(* IEC 61131-3 sources: AXOpen/src/io/ctrl/src, 12 files *)

(* ---- ComponentAvailability.st ---- *)
NAMESPACE AXOpen.Io
    TYPE ComponentAvailability : UINT (
        Available	            :=  UINT#0,	// Hardware component is available.
        ApplicationReadyPending	:=  UINT#1,	// Application Ready Pending; no I/O access.
        LockedBySuperordinated	:=  UINT#2,	// Locked by Superordinated; no access to hardware component.
        LockedByIOController	:=  UINT#3,	// Locked by IO controller; no access to hardware component.
        LockedByIOSupervisor	:=  UINT#4	// Locked by IO supervisor; no access to hardware component.
    );
    END_TYPE
END_NAMESPACE

(* ---- ComponentState.st ---- *)
NAMESPACE AXOpen.Io
    TYPE ComponentState  : UINT (
        Good                    :=	UINT#0, //	No problems detected.
        Disabled                :=	UINT#1, //	The hardware component is disabled.
        MaintenanceRequired     :=	UINT#2, //	Maintenance required.
        MaintenanceDemanded     :=	UINT#3, //	Maintenance demanded.
        Error                   :=	UINT#4, //	Error.
        NotAccessible           :=	UINT#5, //	Status unknown or error in higher-level hardware component.
        Unknown                 :=	UINT#6, //	Default value for components that do not return diagnostic events.
        IONotAvailable          :=	UINT#7  //	Inputs/outputs are not available.
                    );
    END_TYPE
END_NAMESPACE

(* ---- GetDiagnosticsReturnCode.st ---- *)
NAMESPACE AXOpen.Io
    TYPE GetDiagnosticsReturnCode : INT (
        Unknown             :=	INT#-1,     //
        NoError             :=	INT#0,      //	No error.
        HardwareIDInvalid   :=	INT#-32642, //	The address is unknown.
        HardwareIDisInvalid   :=	INT#-32624, //	The address is unknown.
        OutOfResources      :=	INT#-32575  //	All diagnostic resources are currently in use
        ) := Unknown;
    END_TYPE
END_NAMESPACE

(* ---- OperatingState .st ---- *)
NAMESPACE AXOpen.Io
    TYPE OperatingState   : UINT (
        NotSupported                :=	UINT#0,     //	Not Supported; for I/O modules OperatingState always has this value.
        StopFirmwareUpdate          :=	UINT#1,     //	STOP; firmware update.
        StopMemoryReset             :=	UINT#2,     //	STOP; memory reset.
        StopSelfStart               :=	UINT#3,     //	STOP; self start.
        Stop                        :=	UINT#4,     //	STOP.
        MemoryReset                 :=	UINT#5,     //	Memory reset.
        Startup                     :=	UINT#6,     //	STARTUP.
        Run                         :=	UINT#8,     //	RUN.
        RunRedundant                :=	UINT#9,     //	RUN-REDUNDANT.
        Hold                        :=	UINT#10,    //	HOLD.
        Defect                      :=	UINT#13,    //	DEFECT (can only be seen in diagnostic buffer entries).
        DeEnergized                 :=	UINT#15,    //	De-energized (can only be seen in diagnostic buffer entries).
        ConfigurationInRun          :=	UINT#16,    //	Configuration in Run (CiR).
        StopWithoutOutputDisable    :=	UINT#17,    //	STOP without output disable.
        RunWithOutputDisable        :=	UINT#18,    //	RUN with output disable.
        PgmTest                     :=	UINT#19,    //	PgmTest.
        PrimaryRunBackupTest        :=	UINT#20,    //	RunPgmTest (state of primary PLC when the backup PLC is in test mode).
        PrimarySyncup               :=	UINT#21,    //	RUN-SYNCUP (only primary PLC in SYNCUP system state).
        BackupSyncup                :=	UINT#22,    //	SYNCUP (only backup PLC in SYNCUP system state)
        PartnerPlcStateUnknown      :=	UINT#31,    //	State of partner PLC unknown (for example when the partner PLC is not available).
        StopSystemState             :=	UINT#33,    //	STOP system state
        StartupSystemState          :=	UINT#35,    //	STARTUP system state
        RunSoloSystemState          :=	UINT#37,    //	RUN-SOLO system state
        SyncupSystemState           :=	UINT#38,    //	SYNCUP system state
        RunRedundantSystemState     :=	UINT#40    //	RUN-REDUNDANT system state
                    );
    END_TYPE
END_NAMESPACE

(* ---- ReplacementState .st ---- *)
NAMESPACE AXOpen.Io
    TYPE ReplacementState  : UINT (
        Unknown         :=	UINT#255,
        OK              :=	UINT#0, //	The correct element exists.
        Substitute      :=	UINT#1, //	The element was replaced by a compatible element.
        Incompatible    :=	UINT#2, //	The element was replaced by an incompatible element (is reachable, but not ready for operation).
        Missing         :=	UINT#3 //	The element does not exist.
            ) := Unknown;
    END_TYPE
END_NAMESPACE

(* ---- AxoHardwareDiagnostics.st ---- *)
USING AXOpen.Core;
USING AXOpen.Core;
USING AXOpen.Messaging;
USING AXOpen.Messaging.Static;
USING Siemens.Simatic.Diagnostics.Hardware;

NAMESPACE AXOpen.Io
    {S7.extern=ReadWrite}
    CLASS AxoHardwareDiagnostics EXTENDS AXOpen.Core.AxoTask
        VAR PUBLIC
            {#ix-attr:[Container(Layout.Stack)]}
            {#ix-set:AttributeName = "<#Hardware ID#>"}
            {#ix-attr:[ReadOnly()]}
            hardwareID	                :   UINT;	                //  Input	Hardware identifier of the component.
            {#ix-set:AttributeName = "<#Diagnostics return code#>"}
            {#ix-attr:[ReadOnly()]}
            GetDiagnosticsReturnCode    :   GetDiagnosticsReturnCode;
            {#ix-attr:[Container(Layout.Wrap)]}
            {#ix-set:AttributeName = "<#Diagnostics details#>"}
            {#ix-attr:[ReadOnly()]}
            diagnosticDetails	        :   DiagnosticDetails;	    //  Diagnostic information of the addressed hardware component.
        END_VAR

        ///<summary>
        /// Runs tasks and logic of this component.
        /// >[!IMPORTANT] This method must or one of its overloads be called cyclically.
        ///</summary>
        METHOD PUBLIC Run
            VAR_INPUT
                inParent    :   IAxoObject;
                hwID        :   UINT;
            END_VAR
            VAR
                diagInfo : Siemens.Simatic.Diagnostics.Hardware.DiagnosticDetails;
            END_VAR

            IF SUPER.Execute(inParent) THEN
                GetDiagnosticsReturnCode := GetDiagnostics(hwID, diagInfo);

                IF GetDiagnosticsReturnCode=GetDiagnosticsReturnCode#NoError THEN
                    diagnosticDetails.ComponentStateDetail.HardwareComponentState.NoAdditionalInformation   :=  diagInfo.ComponentStateDetail.HardwareComponentState.NoAdditionalInformation;
                    diagnosticDetails.ComponentStateDetail.HardwareComponentState.TransferNotPermitted      :=  diagInfo.ComponentStateDetail.HardwareComponentState.TransferNotPermitted;
                    diagnosticDetails.ComponentStateDetail.HardwareComponentState.DiagnosticsAvailable      :=  diagInfo.ComponentStateDetail.HardwareComponentState.DiagnosticsAvailable;
                    diagnosticDetails.ComponentStateDetail.HardwareComponentState.MaintenanceRequired       :=  diagInfo.ComponentStateDetail.HardwareComponentState.MaintenanceRequired;
                    diagnosticDetails.ComponentStateDetail.HardwareComponentState.MaintenanceDemanded       :=  diagInfo.ComponentStateDetail.HardwareComponentState.MaintenanceDemanded;
                    diagnosticDetails.ComponentStateDetail.HardwareComponentState.Error                     :=  diagInfo.ComponentStateDetail.HardwareComponentState.Error;
                    diagnosticDetails.ComponentStateDetail.HardwareComponentState.ComponentAvailability     :=  diagInfo.ComponentStateDetail.HardwareComponentState.ComponentAvailability;
                    diagnosticDetails.ComponentStateDetail.HardwareComponentState.ReplacementState          :=  diagInfo.ComponentStateDetail.HardwareComponentState.ReplacementState;

                    diagnosticDetails.ComponentStateDetail.PlcState.ModuleDisabled                          :=  diagInfo.ComponentStateDetail.PlcState.ModuleDisabled;
                    diagnosticDetails.ComponentStateDetail.PlcState.ConfigurationInRunActive                :=  diagInfo.ComponentStateDetail.PlcState.ConfigurationInRunActive;
                    diagnosticDetails.ComponentStateDetail.PlcState.InputNotAvailable                       :=  diagInfo.ComponentStateDetail.PlcState.InputNotAvailable;
                    diagnosticDetails.ComponentStateDetail.PlcState.OutputNotAvailable                      :=  diagInfo.ComponentStateDetail.PlcState.OutputNotAvailable;
                    diagnosticDetails.ComponentStateDetail.PlcState.DiagnosticsBufferOverflow               :=  diagInfo.ComponentStateDetail.PlcState.DiagnosticsBufferOverflow;
                    diagnosticDetails.ComponentStateDetail.PlcState.DiagnosticsNotAvailable                 :=  diagInfo.ComponentStateDetail.PlcState.DiagnosticsNotAvailable;
                    diagnosticDetails.ComponentStateDetail.PlcState.PartialDeviceFailure                    :=  diagInfo.ComponentStateDetail.PlcState.PartialDeviceFailure;

                    diagnosticDetails.ComponentState                                                        :=  diagInfo.ComponentState;

                    diagnosticDetails.IoState.Good                                                          :=  diagInfo.IoState.Good;
                    diagnosticDetails.IoState.Disabled                                                      :=  diagInfo.IoState.Disabled;
                    diagnosticDetails.IoState.MaintenanceRequired                                           :=  diagInfo.IoState.MaintenanceRequired;
                    diagnosticDetails.IoState.MaintenanceDemanded                                           :=  diagInfo.IoState.MaintenanceDemanded;
                    diagnosticDetails.IoState.Error                                                         :=  diagInfo.IoState.Error;
                    diagnosticDetails.IoState.NotAccessible                                                 :=  diagInfo.IoState.NotAccessible;
                    diagnosticDetails.IoState.DiagnosticsAvailable                                          :=  diagInfo.IoState.DiagnosticsAvailable;
                    diagnosticDetails.IoState.IODataNotAvailable                                            :=  diagInfo.IoState.IODataNotAvailable;
                    diagnosticDetails.IoState.NetworkError                                                  :=  diagInfo.IoState.NetworkError;
                    diagnosticDetails.IoState.HardwareError                                                 :=  diagInfo.IoState.HardwareError;

                    diagnosticDetails.OperatingState                                                        :=  diagInfo.OperatingState;
                END_IF;

                SUPER.DoneWhen(Duration >= T#500ms AND GetDiagnosticsReturnCode=GetDiagnosticsReturnCode#NoError);
                SUPER.ThrowWhen(Duration >= T#2s OR GetDiagnosticsReturnCode=GetDiagnosticsReturnCode#HardwareIDInvalid OR GetDiagnosticsReturnCode=GetDiagnosticsReturnCode#OutOfResources);
            END_IF;

            IF SUPER.StartTriggered() THEN
                hardwareID := hwID;
                GetDiagnosticsReturnCode                                                                :=  GetDiagnosticsReturnCode#Unknown;

                diagnosticDetails.ComponentStateDetail.HardwareComponentState.NoAdditionalInformation   :=  FALSE;
                diagnosticDetails.ComponentStateDetail.HardwareComponentState.TransferNotPermitted      :=  FALSE;
                diagnosticDetails.ComponentStateDetail.HardwareComponentState.DiagnosticsAvailable      :=  FALSE;
                diagnosticDetails.ComponentStateDetail.HardwareComponentState.MaintenanceRequired       :=  FALSE;
                diagnosticDetails.ComponentStateDetail.HardwareComponentState.MaintenanceDemanded       :=  FALSE;
                diagnosticDetails.ComponentStateDetail.HardwareComponentState.Error                     :=  FALSE;
                diagnosticDetails.ComponentStateDetail.HardwareComponentState.ComponentAvailability     :=  ComponentAvailability#Unknown;
                diagnosticDetails.ComponentStateDetail.HardwareComponentState.ReplacementState          :=  ReplacementState#Unknown;

                diagnosticDetails.ComponentStateDetail.PlcState.ModuleDisabled                          :=  FALSE;
                diagnosticDetails.ComponentStateDetail.PlcState.ConfigurationInRunActive                :=  FALSE;
                diagnosticDetails.ComponentStateDetail.PlcState.InputNotAvailable                       :=  FALSE;
                diagnosticDetails.ComponentStateDetail.PlcState.OutputNotAvailable                      :=  FALSE;
                diagnosticDetails.ComponentStateDetail.PlcState.DiagnosticsBufferOverflow               :=  FALSE;
                diagnosticDetails.ComponentStateDetail.PlcState.DiagnosticsNotAvailable                 :=  FALSE;
                diagnosticDetails.ComponentStateDetail.PlcState.PartialDeviceFailure                    :=  FALSE;

                diagnosticDetails.ComponentState                                                        :=  ComponentState#Unknown;

                diagnosticDetails.IoState.Good                                                          :=  FALSE;
                diagnosticDetails.IoState.Disabled                                                      :=  FALSE;
                diagnosticDetails.IoState.MaintenanceRequired                                           :=  FALSE;
                diagnosticDetails.IoState.MaintenanceDemanded                                           :=  FALSE;
                diagnosticDetails.IoState.Error                                                         :=  FALSE;
                diagnosticDetails.IoState.NotAccessible                                                 :=  FALSE;
                diagnosticDetails.IoState.DiagnosticsAvailable                                          :=  FALSE;
                diagnosticDetails.IoState.IODataNotAvailable                                            :=  FALSE;
                diagnosticDetails.IoState.NetworkError                                                  :=  FALSE;
                diagnosticDetails.IoState.HardwareError                                                 :=  FALSE;

                diagnosticDetails.OperatingState                                                        :=  OperatingState#Unknown;
            END_IF;
        END_METHOD
    END_CLASS
END_NAMESPACE

(* ---- AxoIoComponent.st ---- *)
USING AXOpen.Core;
USING AXOpen.Messaging;
USING AXOpen.Messaging.Static;
USING Siemens.Simatic.S71500.Diagnostics.Hardware;

NAMESPACE AXOpen.Io
    {S7.extern=ReadWrite}
    CLASS AxoIoComponent EXTENDS AXOpen.Core.AxoComponent
        VAR PUBLIC
            {#ix-attr:[Container(Layout.Wrap)]}
            {#ix-attr:[ComponentDetails("Hardware diagnostics")]}
            {#ix-set:AttributeName = "<#Update diagnostics#>"}
            UpdateHardwareDiagnosticsTask : AXOpen.Core.AxoTask;
            {#ix-attr:[ComponentDetails("Hardware diagnostics")]}
            {#ix-attr:[ReadOnly()]}
            {#ix-set:AttributeName = "<#Hardware ID#>"}
            hardwareID	                :   UINT;	                //  Input	Hardware identifier of the component.
            {#ix-attr:[ComponentDetails("Hardware diagnostics")]}
            {#ix-attr:[ReadOnly()]}
            {#ix-set:AttributeName = "<#Diagnostics return code#>"}
            GetDiagnosticsReturnCode    :   GetDiagnosticsReturnCode;
            {#ix-attr:[ComponentDetails("Hardware diagnostics")]}
            {#ix-attr:[ReadOnly()]}
            {#ix-set:AttributeName = "<#Diagnostics details#>"}
            diagnosticDetails	        :   DiagnosticDetails;	    //  Diagnostic information of the addressed hardware component.
        END_VAR

        ///<summary>
        /// Runs tasks and logic of this component.
        /// >[!IMPORTANT] This method must or one of its overloads be called cyclically.
        ///</summary>
        METHOD PUBLIC Run
            VAR_INPUT
                parent  : IAxoObject;
                hwID    :   WORD;
            END_VAR
            IF (parent = NULL) THEN RETURN; END_IF;
            THIS.Initialize(parent);
            THIS.Execute(hwID);
        END_METHOD

        // ///<summary>
        // /// Runs tasks and logic of this component.
        // /// >[!IMPORTANT] This method must or one of its overloads be called cyclically.
        // ///</summary>
        // METHOD PUBLIC Run
        //     VAR_INPUT
        //         parent  : IAxoContext;
        //         hwID    :   WORD;
        //     END_VAR
        //     THIS.Initialize(parent);
        //     THIS.Execute(hwID);
        // END_METHOD

        METHOD PRIVATE Execute
            VAR_INPUT
                hwID    :   WORD;
            END_VAR
            VAR
                diagInfo : Siemens.Simatic.S71500.Diagnostics.Hardware.DiagnosticDetails;
            END_VAR

            UpdateHardwareDiagnosticsTask.Initialize(THIS);

            IF UpdateHardwareDiagnosticsTask.Execute() THEN
                GetDiagnosticsReturnCode := GetDiagnostics(TO_UINT(hwID), diagInfo);
                UpdateHardwareDiagnosticsTask.DoneWhen(UpdateHardwareDiagnosticsTask.Duration >= T#250ms AND GetDiagnosticsReturnCode=GetDiagnosticsReturnCode#NoError);
                UpdateHardwareDiagnosticsTask.ThrowWhen(UpdateHardwareDiagnosticsTask.Duration >= T#250ms AND GetDiagnosticsReturnCode<>GetDiagnosticsReturnCode#NoError);
            END_IF;

            IF UpdateHardwareDiagnosticsTask.DoneReached() THEN
                diagnosticDetails.ComponentStateDetail.HardwareComponentState.NoAdditionalInformation   :=  diagInfo.ComponentStateDetail.HardwareComponentState.NoAdditionalInformation;
                diagnosticDetails.ComponentStateDetail.HardwareComponentState.TransferNotPermitted      :=  diagInfo.ComponentStateDetail.HardwareComponentState.TransferNotPermitted;
                diagnosticDetails.ComponentStateDetail.HardwareComponentState.DiagnosticsAvailable      :=  diagInfo.ComponentStateDetail.HardwareComponentState.DiagnosticsAvailable;
                diagnosticDetails.ComponentStateDetail.HardwareComponentState.MaintenanceRequired       :=  diagInfo.ComponentStateDetail.HardwareComponentState.MaintenanceRequired;
                diagnosticDetails.ComponentStateDetail.HardwareComponentState.MaintenanceDemanded       :=  diagInfo.ComponentStateDetail.HardwareComponentState.MaintenanceDemanded;
                diagnosticDetails.ComponentStateDetail.HardwareComponentState.Error                     :=  diagInfo.ComponentStateDetail.HardwareComponentState.Error;
                diagnosticDetails.ComponentStateDetail.HardwareComponentState.ComponentAvailability     :=  diagInfo.ComponentStateDetail.HardwareComponentState.ComponentAvailability;
                diagnosticDetails.ComponentStateDetail.HardwareComponentState.ReplacementState          :=  diagInfo.ComponentStateDetail.HardwareComponentState.ReplacementState;

                diagnosticDetails.ComponentStateDetail.PlcState.ModuleDisabled                          :=  diagInfo.ComponentStateDetail.PlcState.ModuleDisabled;
                diagnosticDetails.ComponentStateDetail.PlcState.ConfigurationInRunActive                :=  diagInfo.ComponentStateDetail.PlcState.ConfigurationInRunActive;
                diagnosticDetails.ComponentStateDetail.PlcState.InputNotAvailable                       :=  diagInfo.ComponentStateDetail.PlcState.InputNotAvailable;
                diagnosticDetails.ComponentStateDetail.PlcState.OutputNotAvailable                      :=  diagInfo.ComponentStateDetail.PlcState.OutputNotAvailable;
                diagnosticDetails.ComponentStateDetail.PlcState.DiagnosticsBufferOverflow               :=  diagInfo.ComponentStateDetail.PlcState.DiagnosticsBufferOverflow;
                diagnosticDetails.ComponentStateDetail.PlcState.DiagnosticsNotAvailable                 :=  diagInfo.ComponentStateDetail.PlcState.DiagnosticsNotAvailable;
                diagnosticDetails.ComponentStateDetail.PlcState.PartialDeviceFailure                    :=  diagInfo.ComponentStateDetail.PlcState.PartialDeviceFailure;

                diagnosticDetails.ComponentState                                                        :=  diagInfo.ComponentState;

                diagnosticDetails.IoState.Good                                                          :=  diagInfo.IoState.Good;
                diagnosticDetails.IoState.Disabled                                                      :=  diagInfo.IoState.Disabled;
                diagnosticDetails.IoState.MaintenanceRequired                                           :=  diagInfo.IoState.MaintenanceRequired;
                diagnosticDetails.IoState.MaintenanceDemanded                                           :=  diagInfo.IoState.MaintenanceDemanded;
                diagnosticDetails.IoState.Error                                                         :=  diagInfo.IoState.Error;
                diagnosticDetails.IoState.NotAccessible                                                 :=  diagInfo.IoState.NotAccessible;
                diagnosticDetails.IoState.DiagnosticsAvailable                                          :=  diagInfo.IoState.DiagnosticsAvailable;
                diagnosticDetails.IoState.IODataNotAvailable                                            :=  diagInfo.IoState.IODataNotAvailable;
                diagnosticDetails.IoState.NetworkError                                                  :=  diagInfo.IoState.NetworkError;
                diagnosticDetails.IoState.HardwareError                                                 :=  diagInfo.IoState.HardwareError;

                diagnosticDetails.OperatingState                                                        :=  diagInfo.OperatingState;
            END_IF;
        END_METHOD

        METHOD PROTECTED OVERRIDE ManualControl
            THIS._isManuallyControllable := true;
        END_METHOD

        ///<summary>
        /// Restores this component into intial state.
        ///</summary>
        METHOD PUBLIC OVERRIDE Restore
            UpdateHardwareDiagnosticsTask.Restore();
        END_METHOD
    END_CLASS
END_NAMESPACE

(* ---- ComponentStateDetail.st ---- *)
NAMESPACE AXOpen.Io
    {S7.extern=ReadWrite}
    CLASS ComponentStateDetail
        VAR PUBLIC
            HardwareComponentState  :   HardwareComponentState;  //	Represents detailed state information about the hardware component.
            PlcState                :	PlcState;                //	Represents detailed state information about the PLC.
        END_VAR
    END_CLASS
END_NAMESPACE

(* ---- DiagnosticDetails .st ---- *)
NAMESPACE AXOpen.Io
    {S7.extern=ReadWrite}
    CLASS DiagnosticDetails
        VAR PUBLIC
            {#ix-attr:[Container(Layout.Wrap)]}
            {#ix-attr:[Group(GroupLayout.GroupBox)]}
            {#ix-set:AttributeName = "<#Component state details#>"}
            ComponentStateDetail    :	ComponentStateDetail;	//  Represents detailed state information about the hardware component and the PLC.
            {#ix-attr:[Container(Layout.Wrap)]}
            {#ix-attr:[Group(GroupLayout.GroupBox)]}
            {#ix-set:AttributeName = "<#Component state#>"}
            ComponentState          :	ComponentState;	        //  State of the component.
            {#ix-attr:[Container(Layout.Wrap)]}
            {#ix-attr:[Group(GroupLayout.GroupBox)]}
            {#ix-set:AttributeName = "<#IO state#>"}
            IOState                 :	IOState;	            //  State of the inputs and outputs of the component.
            {#ix-attr:[Container(Layout.Wrap)]}
            {#ix-attr:[Group(GroupLayout.GroupBox)]}
            {#ix-set:AttributeName = "<#Operating state#>"}
            OperatingState           :	OperatingState;	        //  Operating state of the PLC.
        END_VAR
    END_CLASS
END_NAMESPACE

(* ---- HardwareComponentState.st ---- *)
NAMESPACE AXOpen.Io
    {S7.extern=ReadWrite}
    CLASS HardwareComponentState
        VAR PUBLIC
            {#ix-attr:[Container(Layout.Stack)]}
            NoAdditionalInformation     :	BOOL;	//  No additional information available.
            TransferNotPermitted        :	BOOL;	//  Transfer not permitted.
            DiagnosticsAvailable        :	BOOL;	//  At least one qualified diagnostics is available.
            MaintenanceRequired         :	BOOL;	//  Maintenance required for at least one channel or the component.
            MaintenanceDemanded         :	BOOL;	//  Maintenance demanded for at least one channel or the component.
            Error                       :	BOOL;	//  Error in at least one channel or the component.
            ComponentAvailability	    :   ComponentAvailability;
            ReplacementState	        :   ReplacementState;
        END_VAR
    END_CLASS
END_NAMESPACE

(* ---- IOState .st ---- *)
NAMESPACE AXOpen.Io
    {S7.extern=ReadWrite}
    CLASS IOState
        VAR PUBLIC
            {#ix-attr:[Container(Layout.Stack)]}
            Good                    :	BOOL;   //	No problems detected.
            Disabled                :	BOOL;   //	The hardware component is disabled.
            MaintenanceRequired     :	BOOL;   //	Maintenance required.
            MaintenanceDemanded     :	BOOL;   //	Maintenance demanded.
            Error                   :	BOOL;   //	Error.
            NotAccessible           :	BOOL;   //	Hardware component not reachable; hardware component cannot be accessed.
            DiagnosticsAvailable    :	BOOL;   //	At least one qualified diagnostics is available.
            IODataNotAvailable      :	BOOL;   //	I/O data not available.
            NetworkError            :	BOOL;   //	Network error.
            HardwareError           :	BOOL;   //	Hardware error.
        END_VAR
    END_CLASS
END_NAMESPACE

(* ---- PlcState.st ---- *)
NAMESPACE AXOpen.Io
    {S7.extern=ReadWrite}
    CLASS PlcState
        VAR PUBLIC
            ModuleDisabled              :   BOOL;   //	Submodule or module disabled.
            ConfigurationInRunActive    :   BOOL;   //	Configuration in Run (CiR) operation is active.
            InputNotAvailable           :   BOOL;   //	Input not available.
            OutputNotAvailable          :   BOOL;   //	Output not available.
            DiagnosticsBufferOverflow   :   BOOL;   //	Overflow of diagnostic buffer.
            DiagnosticsNotAvailable     :   BOOL;   //	Diagnostics not available.
            PartialDeviceFailure        :   BOOL;   //	Partial device failure (with PNIO for Shared iDevices).

        END_VAR
    END_CLASS
END_NAMESPACE
